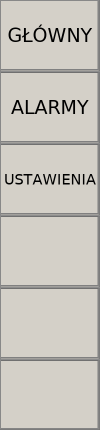
VISUALIZATION MENU_2  // 100x430
    Button (0,0 100x71), "GŁÓWNY", colour toggle: GVL_HMI.hmiPanel.uiNumerEkranu=0
        OnMouseUp: FrameSelectionChange Selection=Selection=-1, GlobSel=IndExpr=0, AssignDir=MAIN.Frames, AssignType=Directly, SelType=Globally
        OnMouseUp: execute { GVL_HMI.hmiPanel.uiMenu	 :=0; GVL_HMI.hmiPanel.bResetMenu := TRUE; }
    Button (0,72 100x71), "ALARMY", colour toggle: GVL_HMI.hmiPanel.uiNumerEkranu=1
        OnMouseUp: FrameSelectionChange Selection=Selection=-1, GlobSel=IndExpr=1, AssignDir=MAIN.Frames, AssignType=Directly, SelType=Globally
        OnMouseUp: execute { GVL_HMI.hmiPanel.uiMenu	 :=1; GVL_HMI.hmiPanel.bResetMenu := TRUE; }
    Button (0,216 100x71)
    Button (0,288 100x71)
    Button (0,360 100x70)
    Button (0,144 100x71), "USTAWIENIA", colour toggle: GVL_HMI.hmiPanel.uiNumerEkranu=2
        OnMouseUp: FrameSelectionChange Selection=Selection=-1, GlobSel=IndExpr=2, AssignDir=MAIN.Frames, AssignType=Directly, SelType=Globally
        OnMouseUp: execute {
            GVL_HMI.hmiPanel.uiMenu	 :=2
            ;
            GVL_HMI.hmiPanel.bResetMenu := TRUE;
        }
END_VISUALIZATION

(* stored: Version 1.1.0.1, ProductVersion 3.1.4024.15
   Visu MENU_2: Id {0c4ffd8c-afe3-4445-9b4b-78b3dabf1a26} *)
